// Mitsubishi GX Works2 project: 시퀀스 부분 반복 연습   PLC: Q03UDV

PROGRAM MAIN
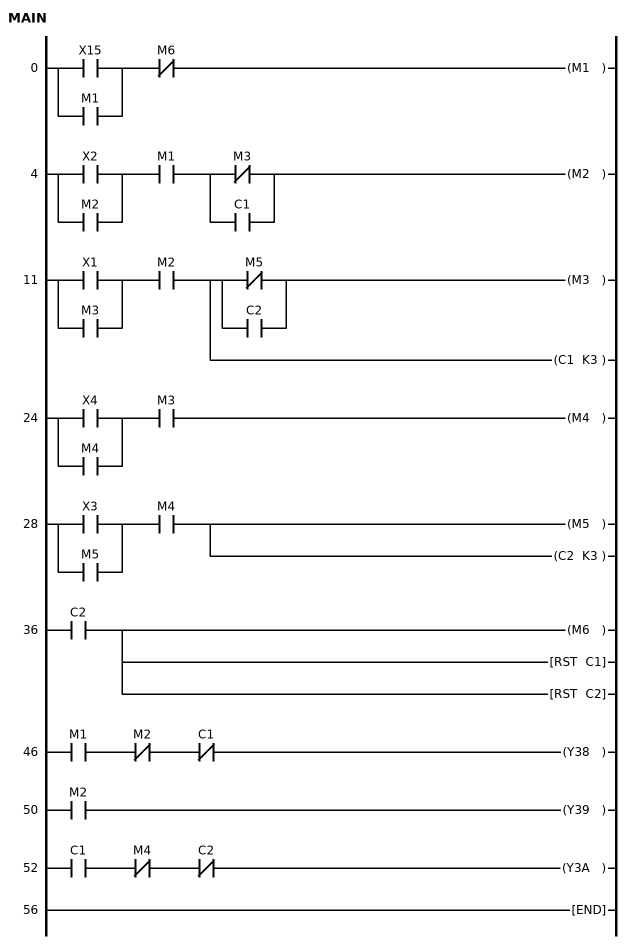
0     LD      X15
      OR      M1
      ANI     M6
      OUT     M1
4     LD      X2
      OR      M2
      AND     M1
      LDI     M3
      OR      C1
      ANB
      OUT     M2
11    LD      X1
      OR      M3
      AND     M2
      MPS
      LDI     M5
      OR      C2
      ANB
      OUT     M3
      MPP
      OUT     C1 K3
24    LD      X4
      OR      M4
      AND     M3
      OUT     M4
28    LD      X3
      OR      M5
      AND     M4
      OUT     M5
      OUT     C2 K3
36    LD      C2
      OUT     M6
      RST     C1
      RST     C2
46    LD      M1
      ANI     M2
      ANI     C1
      OUT     Y38
50    LD      M2
      OUT     Y39
52    LD      C1
      ANI     M4
      ANI     C2
      OUT     Y3A
56    END
END_PROGRAM
